_CFC_ (* Continuous Function Chart, elements in execution order *)
(* 50с *)
#0 AND(TRUE, #11)
#1 YA2_REG_POL <= #0
#2 INT_TO_TIME(SCHU_P2_1_YA2_ZADER_RAS_DOST)
#3 MUL(#2, 1000)
#4 TON_YA2_Rassog1:TON(IN: YA2_DOST, PT: #3)
#5 ABS(SCHU_P2_1_YA2_RASSOG)
#6 GT(#5, SCHU_P2_1_YA2_UST_RASSOG)
#7 AND(NOT SCHU_P2_1_UST_RE_PUSK, #12)
#8 GT(SCHU_P2_1_YA2_RASSOG, SCHU_P2_1_YA2_UST_RASSOG)
#9 SEL(SCHU_P2_1_UST_RE_STOP, #6, #8)
#10 ABS(SCHU_P2_1_YA2_RASSOG_POL)
#11 GT(#10, SCHU_P2_1_YA2_UST_RASSOG)
#12 SEL(YA2_REG_POL, #9, #11)
#13 INT_TO_TIME(SCHU_P2_1_YA2_ZADER_RAS)
#14 MUL(#13, 1000)
#15 TON_YA2_Rassog:TON(IN: #7, PT: #14)
#16 OR(#15.Q, YA2_AO_OTKAZ)
#17 AND(#4.Q, SCHU_P2_1_SA5_DI5_A, #16)
#18 SR_YA2_Otk:SR(SET1: #17, RESET: SCHU_P2_1_SB)
#19 SCHU_P2_1_Z_YA2_OTKAZ <= #18.Q1
_END_CFC_
(* the same logic as Structured Text *)
(* 50с *)
YA2_REG_POL := TRUE AND _t14;
TON_YA2_Rassog1(IN := YA2_DOST, PT := INT_TO_TIME(SCHU_P2_1_YA2_ZADER_RAS_DOST) * 1000);
_t140 := NOT SCHU_P2_1_UST_RE_PUSK AND _t84;
_t14 := ABS(SCHU_P2_1_YA2_RASSOG_POL) > SCHU_P2_1_YA2_UST_RASSOG;
_t84 := SEL(YA2_REG_POL, SEL(SCHU_P2_1_UST_RE_STOP, ABS(SCHU_P2_1_YA2_RASSOG) > SCHU_P2_1_YA2_UST_RASSOG, SCHU_P2_1_YA2_RASSOG > SCHU_P2_1_YA2_UST_RASSOG), _t14);
TON_YA2_Rassog(IN := _t140, PT := INT_TO_TIME(SCHU_P2_1_YA2_ZADER_RAS) * 1000);
SR_YA2_Otk(SET1 := TON_YA2_Rassog1.Q AND SCHU_P2_1_SA5_DI5_A AND (TON_YA2_Rassog.Q OR YA2_AO_OTKAZ), RESET := SCHU_P2_1_SB);
SCHU_P2_1_Z_YA2_OTKAZ := SR_YA2_Otk.Q1;
END_PROGRAM

(* POU TZBiS/TZB/Z_YA3_Otk, CFC *)
PROGRAM Z_YA3_Otk
VAR
	SR_YA3_Otk: SR;
	TON_YA3_Zakl: TON;
	TON_YA3_Rassog: TON;
END_VAR
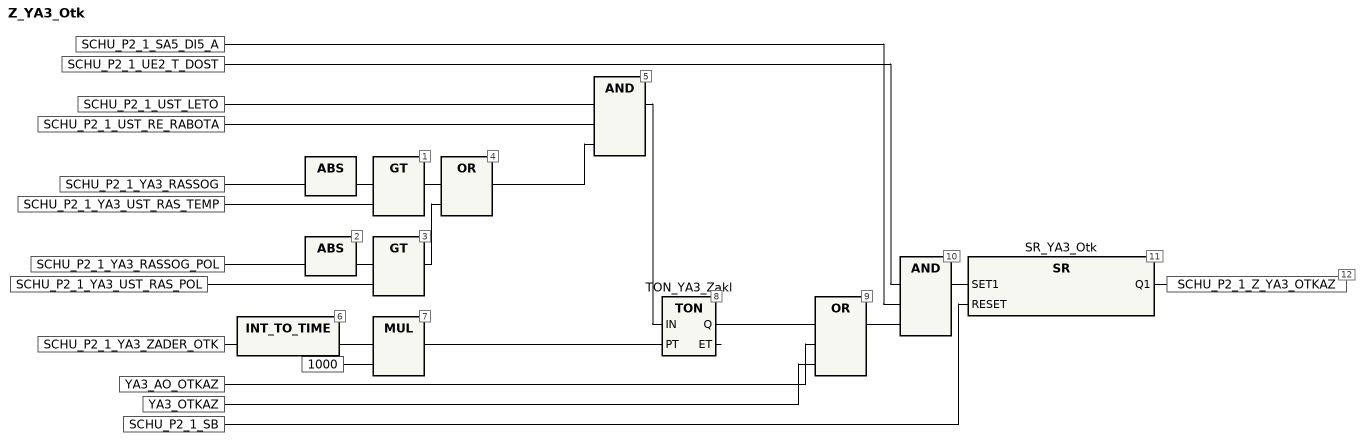
_CFC_ (* Continuous Function Chart, elements in execution order *)
#0 ABS(SCHU_P2_1_YA3_RASSOG)
#1 GT(#0, SCHU_P2_1_YA3_UST_RAS_TEMP)
#2 ABS(SCHU_P2_1_YA3_RASSOG_POL)
#3 GT(#2, SCHU_P2_1_YA3_UST_RAS_POL)
#4 OR(#1, #3)
#5 AND(SCHU_P2_1_UST_LETO, SCHU_P2_1_UST_RE_RABOTA, #4)
#6 INT_TO_TIME(SCHU_P2_1_YA3_ZADER_OTK)
#7 MUL(#6, 1000)
#8 TON_YA3_Zakl:TON(IN: #5, PT: #7)
#9 OR(#8.Q, YA3_AO_OTKAZ, YA3_OTKAZ)
#10 AND(SCHU_P2_1_UE2_T_DOST, SCHU_P2_1_SA5_DI5_A, #9)
#11 SR_YA3_Otk:SR(SET1: #10, RESET: SCHU_P2_1_SB)
#12 SCHU_P2_1_Z_YA3_OTKAZ <= #11.Q1
_END_CFC_
(* the same logic as Structured Text *)
TON_YA3_Zakl(IN := SCHU_P2_1_UST_LETO AND SCHU_P2_1_UST_RE_RABOTA AND ((ABS(SCHU_P2_1_YA3_RASSOG) > SCHU_P2_1_YA3_UST_RAS_TEMP) OR (ABS(SCHU_P2_1_YA3_RASSOG_POL) > SCHU_P2_1_YA3_UST_RAS_POL)), PT := INT_TO_TIME(SCHU_P2_1_YA3_ZADER_OTK) * 1000);
SR_YA3_Otk(SET1 := SCHU_P2_1_UE2_T_DOST AND SCHU_P2_1_SA5_DI5_A AND (TON_YA3_Zakl.Q OR YA3_AO_OTKAZ OR YA3_OTKAZ), RESET := SCHU_P2_1_SB);
SCHU_P2_1_Z_YA3_OTKAZ := SR_YA3_Otk.Q1;
END_PROGRAM

(* POU TZBiS/TZB/Z_YA4_Otk, CFC *)
PROGRAM Z_YA4_Otk
VAR
	RS_YA4_OTKZ: SR;

	UE3_ZADER: TON;
	SCHU_P2_1_YA4_AO4ER: TON;
	F_trig_ai: F_TRIG;
	TON_YA4: TON;
	YA4_ZADER_POL: TON;
	YA4_ZADER_TEMP: TON;
END_VAR
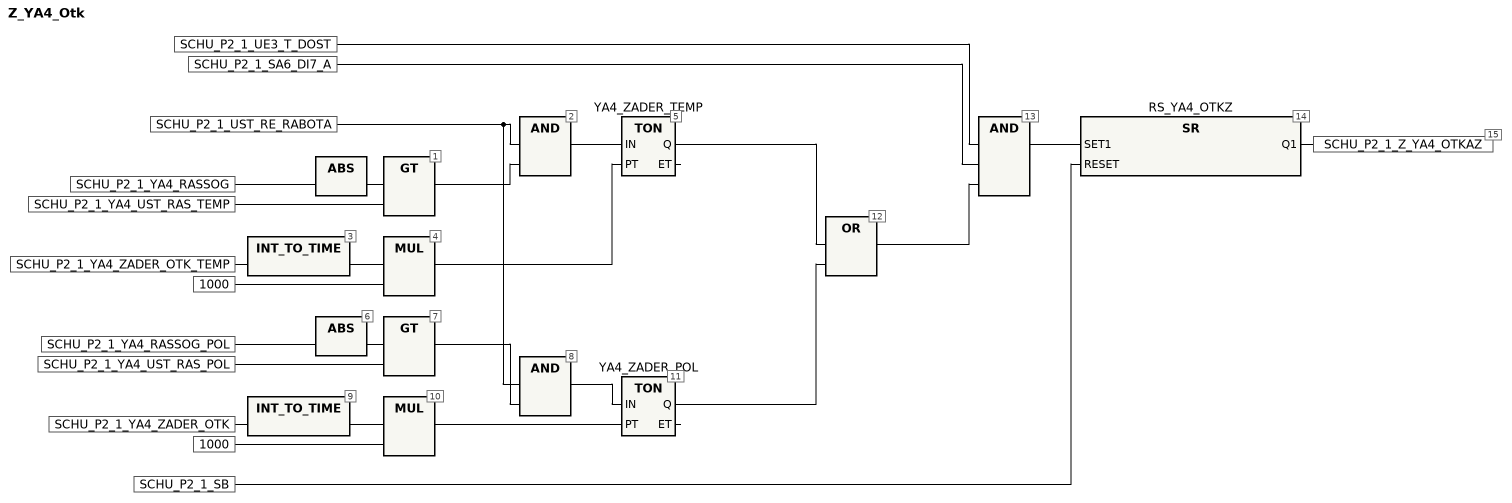
